Staubli VAL3: toJointRxDeg.pgx

public program toJointRxDeg(num& x_nJointArray[], jointRx& x_jJointRx)
  local num l_nRad2Deg
begin
  // Copyright (c) 2016, Ocado Technology - Robotics Research Team
  //
  // Licensed under the Apache License, Version 2.0 (the "License");
  // you may not use this file except in compliance with the License.
  // You may obtain a copy of the License at
  //
  //     http://www.apache.org/licenses/LICENSE-2.0
  //
  // Unless required by applicable law or agreed to in writing, software
  // distributed under the License is distributed on an "AS IS" BASIS,
  // WITHOUT WARRANTIES OR CONDITIONS OF ANY KIND, either express or implied.
  // See the License for the specific language governing permissions and
  // limitations under the License.



  l_nRad2Deg = 57.2957795131

  x_jJointRx.j1 = x_nJointArray[0]
  x_jJointRx.j2 = x_nJointArray[1]
  x_jJointRx.j3 = x_nJointArray[2]
  x_jJointRx.j4 = x_nJointArray[3]
  x_jJointRx.j5 = x_nJointArray[4]
  x_jJointRx.j6 = x_nJointArray[5]
  // popUpMsg("Axes: "+toString(".6", x_jJointRx.j1)+","+toString(".6", x_jJointRx.j2)+","+toString(".6", x_jJointRx.j3)+","+toString(".6", x_jJointRx.j4)+","+toString(".6", x_jJointRx.j5)+","+toString(".6", x_jJointRx.j6))
end
